# EPICS autosave request: iocBoot/iocTest/auto_settings.req
file "quadEM_settings.req",            P=$(P), R=QE1:
file "quadEM_TimeSeries_settings.req", P=$(P), R=QE1_TS:
